{attribute 'GeneratedUsingTerminal: ELX3181-0000-0016'}
{attribute addProperty BoxType "ELX3181-0000-0016"}
{attribute addProperty Id "AdsAddrAT %I*.TcoAmsAddr0AoeNetIdAT %I*.TcoAmsNetId0StateAT %I*UINT2"}
{attribute addProperty CRC "1103447971"}
{attribute addProperty Size "2"}
TYPE InfoData_41C547A3 :
STRUCT
	{attribute addProperty Name "AdsAddr"}
	AdsAddr AT %I* : .TcoAmsAddr;
	{attribute addProperty Name "AoeNetId"}
	AoeNetId AT %I* : .TcoAmsNetId;
	{attribute addProperty Name "State"}
	State AT %I* : UINT;
END_STRUCT
END_TYPE

(* stored: Version 1.2.0.0, ProductVersion 3.1.4024.9
   DUT InfoData_41C547A3: Id {5916a0b4-9ceb-4937-acf6-91649529676c} *)
